// TIA Portal V17 export
// export: Created 2021-11-12T21:16:16.2252169Z, ExportSetting WithDefaults, DisplayName Totally Integrated Automation Portal, DisplayVersion V17 Update 1, DisplayName TIA Portal Openness, DisplayVersion V17 Update 1, DisplayName TIA Portal Version Control Interface, DisplayVersion V17, DisplayName SINAMICS Startdrive Advanced, DisplayVersion V17 Update1, DisplayName SINAMICS Startdrive G110M, G120, G120C, G120D, G120P, G115D, DisplayVersion V17 Update1, DisplayName SINAMICS Startdrive G130, G150, S120, S150, SINAMICS MV, S210, DisplayVersion V17 Update1, DisplayName STEP 7 Professional, DisplayVersion V17 Update 1, DisplayName STEP 7 Safety, DisplayVersion V17, DisplayName WinCC Advanced, DisplayVersion V17 Update 1
DATA_BLOCK "DB - 1 - Modbus Danfoss - MB-01"   // DB7
// stored: AutoNumber true, InstanceOfName FB - 1 - Modbus Danfoss - MB-01, InstanceOfType FB
"FB - 1 - Modbus Danfoss - MB-01"
   // VAR_INPUT
   //    FirstScan : Bool;
   //    RW_TCPModBUS_IP_Oct_1_MB : USInt;
   //    RW_TCPModBUS_IP_Oct_2_MB : USInt;
   //    RW_TCPModBUS_IP_Oct_3_MB : USInt;
   //    RW_TCPModBUS_IP_Oct_4_MB : USInt;
   //    RW_MinMotorFreqHz_MB_Hz : UInt;
   //    RW_MaxMotorFreqHz_MB_Hz : UInt;
   // END_VAR
   // VAR_OUTPUT
   //    RO_SomatorioConsumo_kWh : Real;
   //    RO_CorrenteAtual_A : Real;
   //    RO_FrequenciaAtual_Hz : Real;
   //    RO_PotenciaAtual_kW : Real;
   //    RO_TensaoAtualSaida_V : Real;
   //    RO_MotorRPM : Real;
   //    RO_TempDriveDissipadorCalor_C : Real;
   //    RO_TempDriveCartaoControle_C : Real;
   //    RO_HorimetroMotor_H : Real;
   //    RO_HorimetroDrive_H : Real;
   //    RO_UltimoAlarme : Int;
   //    "RO_AnalogInput53_ma-V" : Real;
   //    "RO_AnalogInput54_ma-V" : Real;
   //    Cfg_Potencia_Motor_kW : Real;
   //    Cfg_Motor_hp : Real;
   //    Cfg_Motor_TensaoNominal_V : Real;
   //    Cfg_Corrente_Nominal_A : Real;
   //    Cfg_Velocidade_Nominal_RPM : Real;
   //    RO_Numero_de_PartidasMotor : Real;
   //    RO_Numero_de_PartidasDrive : Real;
   //    RO_TensaoBarramento_DC_V : Real;
   //    RO_TensaoAmpla_V : Real;
   // END_VAR
   // VAR
   //    MB_Mode { ExternalAccessible := 'False'; ExternalVisible := 'False'; ExternalWritable := 'False'} : USInt;
   //    DataLen { ExternalAccessible := 'False'; ExternalVisible := 'False'; ExternalWritable := 'False'} : USInt;
   //    tmp_real { ExternalAccessible := 'False'; ExternalVisible := 'False'; ExternalWritable := 'False'} : Real;
   //    tmp_word { ExternalAccessible := 'False'; ExternalVisible := 'False'; ExternalWritable := 'False'} : Word;
   //    M_DataAddrReq { ExternalAccessible := 'False'; ExternalVisible := 'False'; ExternalWritable := 'False'} : UDInt;
   //    TypeWrite { ExternalAccessible := 'False'; ExternalVisible := 'False'; ExternalWritable := 'False'} : Bool;
   //    Alternate { ExternalAccessible := 'False'; ExternalVisible := 'False'; ExternalWritable := 'False'} : Int;
   //    M_TCPTmpValueDWord { ExternalAccessible := 'False'; ExternalVisible := 'False'; ExternalWritable := 'False'} : DWord;
   //    M_TCPTmpValueUInt { ExternalAccessible := 'False'; ExternalVisible := 'False'; ExternalWritable := 'False'} : UInt;
   // END_VAR
BEGIN
END_DATA_BLOCK
